            6:      // M2c -> T8, T9, T10
                sPayloadTools := CONCAT('{"', arrMachines[iMachIdx]);
                sPayloadTools := CONCAT(sPayloadTools, '_T8_Usage_sec":');
                sPayloadTools := CONCAT(sPayloadTools, UDINT_TO_STRING(arrToolTimePerMachine[iMachIdx, 8]));
                sPayloadTools := CONCAT(sPayloadTools, ',"');
                sPayloadTools := CONCAT(sPayloadTools, arrMachines[iMachIdx]);
                sPayloadTools := CONCAT(sPayloadTools, '_T9_Usage_sec":');
                sPayloadTools := CONCAT(sPayloadTools, UDINT_TO_STRING(arrToolTimePerMachine[iMachIdx, 9]));
                sPayloadTools := CONCAT(sPayloadTools, ',"');
                sPayloadTools := CONCAT(sPayloadTools, arrMachines[iMachIdx]);
                sPayloadTools := CONCAT(sPayloadTools, '_T10_Usage_sec":');
                sPayloadTools := CONCAT(sPayloadTools, UDINT_TO_STRING(arrToolTimePerMachine[iMachIdx, 10]));
                sPayloadTools := CONCAT(sPayloadTools, '}');

            7, 8:   // M3a, M3b -> T4, T5, T6
                sPayloadTools := CONCAT('{"', arrMachines[iMachIdx]);
                sPayloadTools := CONCAT(sPayloadTools, '_T4_Usage_sec":');
                sPayloadTools := CONCAT(sPayloadTools, UDINT_TO_STRING(arrToolTimePerMachine[iMachIdx, 4]));
                sPayloadTools := CONCAT(sPayloadTools, ',"');
                sPayloadTools := CONCAT(sPayloadTools, arrMachines[iMachIdx]);
                sPayloadTools := CONCAT(sPayloadTools, '_T5_Usage_sec":');
                sPayloadTools := CONCAT(sPayloadTools, UDINT_TO_STRING(arrToolTimePerMachine[iMachIdx, 5]));
                sPayloadTools := CONCAT(sPayloadTools, ',"');
                sPayloadTools := CONCAT(sPayloadTools, arrMachines[iMachIdx]);
                sPayloadTools := CONCAT(sPayloadTools, '_T6_Usage_sec":');
                sPayloadTools := CONCAT(sPayloadTools, UDINT_TO_STRING(arrToolTimePerMachine[iMachIdx, 6]));
                sPayloadTools := CONCAT(sPayloadTools, '}');

            9:      // M3c -> T8, T9, T11
                sPayloadTools := CONCAT('{"', arrMachines[iMachIdx]);
                sPayloadTools := CONCAT(sPayloadTools, '_T8_Usage_sec":');
                sPayloadTools := CONCAT(sPayloadTools, UDINT_TO_STRING(arrToolTimePerMachine[iMachIdx, 8]));
                sPayloadTools := CONCAT(sPayloadTools, ',"');
                sPayloadTools := CONCAT(sPayloadTools, arrMachines[iMachIdx]);
                sPayloadTools := CONCAT(sPayloadTools, '_T9_Usage_sec":');
                sPayloadTools := CONCAT(sPayloadTools, UDINT_TO_STRING(arrToolTimePerMachine[iMachIdx, 9]));
                sPayloadTools := CONCAT(sPayloadTools, ',"');
                sPayloadTools := CONCAT(sPayloadTools, arrMachines[iMachIdx]);
                sPayloadTools := CONCAT(sPayloadTools, '_T11_Usage_sec":');
                sPayloadTools := CONCAT(sPayloadTools, UDINT_TO_STRING(arrToolTimePerMachine[iMachIdx, 11]));
                sPayloadTools := CONCAT(sPayloadTools, '}');

            10, 11: // M4a, M4b -> T4, T5, T6
                sPayloadTools := CONCAT('{"', arrMachines[iMachIdx]);
                sPayloadTools := CONCAT(sPayloadTools, '_T4_Usage_sec":');
                sPayloadTools := CONCAT(sPayloadTools, UDINT_TO_STRING(arrToolTimePerMachine[iMachIdx, 4]));
                sPayloadTools := CONCAT(sPayloadTools, ',"');
                sPayloadTools := CONCAT(sPayloadTools, arrMachines[iMachIdx]);
                sPayloadTools := CONCAT(sPayloadTools, '_T5_Usage_sec":');
                sPayloadTools := CONCAT(sPayloadTools, UDINT_TO_STRING(arrToolTimePerMachine[iMachIdx, 5]));
                sPayloadTools := CONCAT(sPayloadTools, ',"');
                sPayloadTools := CONCAT(sPayloadTools, arrMachines[iMachIdx]);
                sPayloadTools := CONCAT(sPayloadTools, '_T6_Usage_sec":');
                sPayloadTools := CONCAT(sPayloadTools, UDINT_TO_STRING(arrToolTimePerMachine[iMachIdx, 6]));
                sPayloadTools := CONCAT(sPayloadTools, '}');

            12:     // M4c -> T8, T9, T10
                sPayloadTools := CONCAT('{"', arrMachines[iMachIdx]);
                sPayloadTools := CONCAT(sPayloadTools, '_T8_Usage_sec":');
                sPayloadTools := CONCAT(sPayloadTools, UDINT_TO_STRING(arrToolTimePerMachine[iMachIdx, 8]));
                sPayloadTools := CONCAT(sPayloadTools, ',"');
                sPayloadTools := CONCAT(sPayloadTools, arrMachines[iMachIdx]);
                sPayloadTools := CONCAT(sPayloadTools, '_T9_Usage_sec":');
                sPayloadTools := CONCAT(sPayloadTools, UDINT_TO_STRING(arrToolTimePerMachine[iMachIdx, 9]));
                sPayloadTools := CONCAT(sPayloadTools, ',"');
                sPayloadTools := CONCAT(sPayloadTools, arrMachines[iMachIdx]);
                sPayloadTools := CONCAT(sPayloadTools, '_T10_Usage_sec":');
                sPayloadTools := CONCAT(sPayloadTools, UDINT_TO_STRING(arrToolTimePerMachine[iMachIdx, 10]));
                sPayloadTools := CONCAT(sPayloadTools, '}');
        END_CASE
        iStep := 40;

    40: // Envia payload da máquina atual e avança
        bExecutePublish := TRUE;
        IF fbMqttPublish.xDone THEN
            bExecutePublish := FALSE;
            iMachIdx := iMachIdx + 1;
            IF iMachIdx > 12 THEN
                iStep := 0;     // Concluído
            ELSE
                iStep := 30;    // Próxima máquina
            END_IF
        ELSIF fbMqttPublish.xError OR NOT fbMqttClient.xConnectedToBroker THEN
            iStep := 0;
        END_IF

END_CASE

// ==========================================
// 6. BLOCO MQTT PUBLISH
//    Steps 10/20 -> sPayload (Tool + Status)
//    Steps 30/40 -> sPayloadTools (tempos por máquina)
// ==========================================
IF iStep = 30 OR iStep = 40 THEN
    fbMqttPublish(
        xExecute       := bExecutePublish,
        mqttClient     := fbMqttClient,
        wsTopicName    := wsTopic,
        pbPayload      := ADR(sPayloadTools),
        udiPayloadSize := INT_TO_UDINT(LEN(sPayloadTools)),
        eQoS           := 0,
        xRetain        := FALSE
    );
ELSE
    fbMqttPublish(
        xExecute       := bExecutePublish,
        mqttClient     := fbMqttClient,
        wsTopicName    := wsTopic,
        pbPayload      := ADR(sPayload),
        udiPayloadSize := INT_TO_UDINT(LEN(sPayload)),
        eQoS           := 0,
        xRetain        := FALSE
    );
END_IF

END_PROGRAM
